// SIMATIC STEP 7 (V5.x) project ZEn01_12_STEP7__Com_SFC2
// program: ProgrammClient(MPI=10) - Example  Communication  SFC XSEND / XRCV
client program
// program: ProgrammServer(MPI=15) - Example communication SFC XSEND / XRCV
server program

SYMBOL_TABLE
"Data_X_SEND-1"	DB 1	DB 1
"Data_X_SEND-2"	DB 2	DB 2
"Data_X_SEND-3"	DB 3	DB 3
"Modify Values"	FC 1	FC 1
"Communication(send)"	FC 10	FC 10
"CYCL_EXC"	OB 1	OB 1	// Cycle Execution
"CYC_INT5"	OB 35	OB 35	// Cyclic Interrupt 5
"COMPLETE RESTART"	OB 100	OB 100	// Complete Restart
"X_SEND"	SFC 65	SFC 65
"X_RCV"	SFC 66	SFC 66
"X_GET"	SFC 67	SFC 67
"X_PUT"	SFC 68	SFC 68
"X_ABORT"	SFC 69	SFC 69
"I_GET"	SFC 72	SFC 72
"I_PUT"	SFC 73	SFC 73
"I_ABORT"	SFC 74	SFC 74
END_SYMBOL_TABLE

FUNCTION "Modify Values" : VOID	// FC 1
TITLE = Function for Generating a Modifiable Date
AUTHOR : SIEMENS
VERSION : 1.0
BEGIN
NETWORK
TITLE = Incrementing and Saving a Value
      L     MD 60;
      L     1;
      +D;
      T     MD 60;
//Save the variables to be sent in a double word
      T     DB1.DBD 0;	//First double word of variable "X_SEND-1".Array10Byte 
      T     "Data_X_SEND-2".DoubleWord;	//Variable "X_SEND-2".DoubleWord
      T     DB3.DBD 0;	//First double word of variable "X_SEND-3".Array3Words
END_FUNCTION

FUNCTION "Communication(send)" : VOID	// FC 10
VERSION : 1.0
BEGIN
NETWORK
TITLE = X_SEND Block Call 
//Query which X_SEND SFC is currently active
      L     MW 50;	//X_SEND SFC variable: "X_SEND-1".Array10Byte (DB1.DBb 0 to 9) 
      L     1;
      ==I;
      JC    m001;	//Jump to SFC X_SEND variable: "X_SEND-1".Array10Byte  
      L     MW 50;	//X_SEND SFC variable: "X_SEND-2".DoubleWord (DB2.DBD 0) 
      L     2;
      ==I;
      JC    m002;	//Jump to X_SEND SFC variable: "X_SEND-2".DoubleWord  
      L     MW 50;	//X_SEND SFC variable: "X_SEND-3".Array3Words (DB1.DBW 0 to 3) 
      L     3;
      ==I;
      JC    m003;	//Jump to X_SEND SFC variable: "X_SEND-3".Array3Words  
      BEU;
m001: CALL  "X_SEND" (
           REQ                      := M 100.2,
           CONT                     := M 100.3,
           DEST_ID                  := MW 110,
           REQ_ID                   := MD 120,
           SD                       := "Data_X_SEND-1".Array10Bytes,
           RET_VAL                  := MW 132,
           BUSY                     := M 100.4);	//Call X_SEND block / Transfer data (Yes/No)? / Maintain connection (Yes/No)? / Address of receiver / Job number / Send data 10 bytes (DB1) / Return value / SFC active?
//Edge evaluation: Is communication with the falling edge of the BUSY bit
//finished?
      A     M 100.4;
      FN    M 100.5;
      JC    m004;	//Jump to increment the communication memory word
      BEU;
m002: CALL  "X_SEND" (
           REQ                      := M 101.2,
           CONT                     := M 101.3,
           DEST_ID                  := MW 112,
           REQ_ID                   := MD 124,
           SD                       := "Data_X_SEND-2".DoubleWord,
           RET_VAL                  := MW 134,
           BUSY                     := M 101.4);	//Call X_SEND block / Transfer data (Yes/No)? / Maintain connection (Yes/No)? / Address of receiver / Job number / Send data 1 double word (DB2) / Return value / SFC active?
//Edge evaluation: Is communication with the falling edge of the BUSY bit
//finished?
      A     M 101.4;
      FN    M 101.5;
      JC    m005;	//Jump to increment the communication memory word
      BEU;
m003: CALL  "X_SEND" (
           REQ                      := M 102.2,
           CONT                     := M 102.3,
           DEST_ID                  := MW 114,
           REQ_ID                   := MD 128,
           SD                       := "Data_X_SEND-3".Array3Words,
           RET_VAL                  := MW 136,
           BUSY                     := M 102.4);	//Call X_SEND block / Transfer data (Yes/No)? / Maintain connection (Yes/No)? / Address of receiver / Job number / Send data 3 words (DB3) / Return value / SFC active?
//Edge evaluation: Is communication with the falling edge of the BUSY bit
//finished?
      A     M 102.4;
      FN    M 102.5;
      JC    m006;	//Jump to increment the communication memory word
      BEU;
//In the following section, the communication counter is incremented following  
//communication.
m004: L     2;	//Increment after sending "X_SEND-1".Array10Byte
      T     MW 50;
      CALL  "Modify Values";	//The values in the variables are incremented
      BEU;
m005: L     3;	//Increment after sending "X_SEND-2".DoubleWord
      T     MW 50;
      CALL  "Modify Values";	//The values in the variables are incremented
      BEU;
m006: L     1;	//Increment after sending "X_SEND-3".Array3Words
      T     MW 50;
      CALL  "Modify Values";	//The values in the variables are incremented
      BEU;
END_FUNCTION

DATA_BLOCK "Data_X_SEND-1"	// DB 1
AUTHOR : SIEMENS
VERSION : 1.0
  STRUCT
   Array10Bytes : ARRAY  [1 .. 10 ] OF //Array of 10 bytes
   BYTE  := 5 (B#16#10) , 5 (B#16#10) ;
  END_STRUCT ;	
BEGIN
   Array10Bytes[1] := B#16#10;
   Array10Bytes[2] := B#16#10;
   Array10Bytes[3] := B#16#10;
   Array10Bytes[4] := B#16#10;
   Array10Bytes[5] := B#16#10;
   Array10Bytes[6] := B#16#10;
   Array10Bytes[7] := B#16#10;
   Array10Bytes[8] := B#16#10;
   Array10Bytes[9] := B#16#10;
   Array10Bytes[10] := B#16#10;
END_DATA_BLOCK

DATA_BLOCK "Data_X_SEND-2"	// DB 2
AUTHOR : SIEMENS
VERSION : 1.0
  STRUCT
   DoubleWord : DWORD  := DW#16#2D;	//Double word
  END_STRUCT ;	
BEGIN
   DoubleWord := DW#16#2D;
END_DATA_BLOCK

DATA_BLOCK "Data_X_SEND-3"	// DB 3
AUTHOR : SIEMENS
VERSION : 1.0
  STRUCT
   Array3Words : ARRAY  [1 .. 3 ] OF //Array of 3 words
   WORD  := 3 (W#16#3) ;
  END_STRUCT ;	
BEGIN
   Array3Words[1] := W#16#3;
   Array3Words[2] := W#16#3;
   Array3Words[3] := W#16#3;
END_DATA_BLOCK

ORGANIZATION_BLOCK "CYCL_EXC"	// OB 1
TITLE = Cyclically Processing Program
AUTHOR : SIEMENS
VERSION : 1.0
VAR_TEMP
  OB1_EV_CLASS : BYTE ;	//Bits 0 to 3 = 1 (incoming event), bits 4 to 7 = 1 (event class 1)
  OB1_SCAN_1 : BYTE ;	//1 (Cold restart scan 1 of OB1), 3 (Scan 2-n of OB1)
  OB1_PRIORITY : BYTE ;	//1 (Priority of 1 is lowest)
  OB1_OB_NUMBR : BYTE ;	//1 (Organization block 1, OB1)
  OB1_RESERVED_1 : BYTE ;	//Reserved for system
  OB1_RESERVED_2 : BYTE ;	//Reserved for system
  OB1_PREV_CYCLE : INT ;	//Cycle time of previous OB1 scan (milliseconds)
  OB1_MIN_CYCLE : INT ;	//Minimum cycle time of OB1 (milliseconds)
  OB1_MAX_CYCLE : INT ;	//Maximum cycle time of OB1 (milliseconds)
  OB1_DATE_TIME : DATE_AND_TIME ;	//Date and time OB1 started
END_VAR
BEGIN
NETWORK
TITLE = Description of the Communication Function 
NETWORK
TITLE = Default Settings for the SFC Parameters
//
//By setting the following 3 memory bits, you can ensure that the connection 
//between 
//the communication partners is retained following each SFC call.
      SET;
      =     M 100.3;	//Connection should be maintained after SFC call 
      =     M 101.3;	//Connection should be maintained after SFC call
      =     M 102.3;	//Connection should be maintained after SFC call 
// Default address for SFCs
      L     15;	//Load MPI subnet address or 
//                                        the address of the logical node number
      T     MW 110;	//SFC call, send an array of 10 bytes (DB1)
      T     MW 112;	//SFC call, send a double word (DB2)
      T     MW 114;	//SFC call, send an array of 3 words (DB3)
//Assignment of the job number
      L     1;	//Load first job number
      T     MD 120;	//Assign to SFC call (array of 10 bytes)
      L     2;	//Load second job number
      T     MD 124;	//Assign to SFC call (double word)
      L     3;	//Load third job number
      T     MD 128;	//Assign to SFC call (array 3 words)
END_ORGANIZATION_BLOCK

ORGANIZATION_BLOCK "CYC_INT5"	// OB 35
TITLE = Call Every 100 ms
AUTHOR : SIEMENS
VERSION : 1.0
VAR_TEMP
  OB35_EV_CLASS : BYTE ;	//Bits 0 to 3 = 1 (incoming event), bits 4 to 7 = 1 (event class 1)
  OB35_STRT_INF : BYTE ;	//16#36 (OB35 has started)
  OB35_PRIORITY : BYTE ;	//11 (Priority of 1 is lowest)
  OB35_OB_NUMBR : BYTE ;	//35 (Organization block 35, OB35)
  OB35_RESERVED_1 : BYTE ;	//Reserved for system
  OB35_RESERVED_2 : BYTE ;	//Reserved for system
  OB35_PHASE_OFFSET : WORD ;	//Phase offset (ms)
  OB35_RESERVED_3 : INT ;	//Reserved for system
  OB35_EXC_FREQ : INT ;	//Frequency of execution (ms)
  OB35_DATE_TIME : DATE_AND_TIME ;	//Date and time OB35 started
END_VAR
BEGIN
NETWORK
TITLE = Communicating with Server S7 Station B
//********************************************************************************
//******************
//General Description of the Communication Function of this Client S7 Station A
//********************************************************************************
//******************
//
//Three variables are exchanged between this client S7-300 station A and the 
//server S7-300 station B. 
//The variable "X_SEND-1".Feld10byte (DB1.DBB 0 to 9) is sent to server MPI 15 
//with the SFC X_SEND.
//An SFC call is required for this.
//The same procedure is required for the variable "X_SEND-2".Doppelwort (DB2.DBD 
//0).
//The variable "X_SEND-1".Feld3Worte (DB3.DBW 0 to 2) is the third variable to be 
//written by the  
//client to a variable of the same name on the server with the SFC X_SEND.
//The variables can be found in DBs 1 to 3 on both the client and the server 
//side. 
//The connection between the communicating CPUs is established the first time an 
//SFC is called 
//and then maintained (only one connection resource is required).
//The SFCs are called by OB35 using a timer in order to make them independent of 
//the 
//scan cycle time of OB1 in the client and the server CPU.
//The timers for the OB calls are preset when the CPU is configured.
//In this CPU, OB35 is called every 100 ms(default), and this means that the 
//various SFCs are also 
//called every 100 ms (max.). 
//Once data exchange is complete, the data are changed in the variables in order 
//to show that  
//data have been received. If there is an error in the communication, and no data 
//are
//sent, the data in the receiver will not change. 
//If the receive data are continually changing, this means that data exchange is 
//taking place. 
//
//
//Note:
//The memory words in which the RET_VALS of the SFCs are entered should be 
//evaluated while the  
//program is running. If an SFC registers an error value, it can still be 
//correctly executed, 
//although no data will have been sent. 
//As soon as the RET_VAL of an SFC becomes negative, this signals that an error 
//has
//occurred during data transmission. 
//
//
//Memory words in which the RET_VALs are entered:
//MW130, MW132, MW134
//
//The above note was not taken into account in this programming example, since 
//error messages 
//which may occur cannot be converted to corresponding messages (alarms which 
//appear on the device) 
//until a real control program is run.
//
      CALL  "Communication(send)";	//Call communication function
END_ORGANIZATION_BLOCK

ORGANIZATION_BLOCK "COMPLETE RESTART"	// OB 100
AUTHOR : SIEMENS
VERSION : 1.0
VAR_TEMP
  OB100_EV_CLASS : BYTE ;	//16#13, Event class 1, entering event state, event logged in diagnostic buffer
  OB100_STRTUP : BYTE ;	//16#81/82/83/84 Method of startup
  OB100_PRIORITY : BYTE ;	//27 (Priority of 1 is lowest)
  OB100_OB_NUMBR : BYTE ;	//100 (Organization block 100, OB100)
  OB100_RESERVED_1 : BYTE ;	//Reserved for system
  OB100_RESERVED_2 : BYTE ;	//Reserved for system
  OB100_STOP : WORD ;	//Event that caused CPU to stop (16#4xxx)
  OB100_STRT_INFO : DWORD ;	//Information on how system started
  OB100_DATE_TIME : DATE_AND_TIME ;	//Date and time OB100 started
END_VAR
BEGIN
NETWORK
TITLE = Initial Value Assignment
      L     1;	//Preset communication memory word
      T     MW 50;
      SET;	//Set starting memory bit of SFC X_SEND   
      =     M 100.2;	//SFC X_SEND variable: "X_SEND-1".Array10Byte
      =     M 101.2;	//SFC X_SEND variable: "X_SEND-2".DoubleWord
      =     M 102.2;	//SFC X_SEND variable: "X_SEND-3".Array3Words
END_ORGANIZATION_BLOCK

SYMBOL_TABLE
"Data_X_RCV-1"	DB 1	DB 1
"Data_X_RCV-2"	DB 2	DB 2
"Data_X_RCV-3"	DB 3	DB 3
"Modify Values"	FC 1	FC 1
"Communication(receive)"	FC 20	FC 20
"CYCL_EXC"	OB 1	OB 1	// Cycle Execution
"CYC_INT5"	OB 35	OB 35	// Cyclic Interrupt 5
"COMPLETE RESTART"	OB 100	OB 100	// Complete Restart
"X_SEND"	SFC 65	SFC 65
"X_RCV"	SFC 66	SFC 66
"X_GET"	SFC 67	SFC 67
"X_PUT"	SFC 68	SFC 68
"X_ABORT"	SFC 69	SFC 69
"I_GET"	SFC 72	SFC 72
"I_PUT"	SFC 73	SFC 73
"I_ABORT"	SFC 74	SFC 74
END_SYMBOL_TABLE

FUNCTION "Communication(receive)" : VOID	// FC 20
TITLE = Receiving Data from Client S7 Station A
AUTHOR : SIEMENS
VERSION : 1.0
VAR_TEMP
  NIL_PTR : ANY ;	//NIL pointer, required in order to discard data
END_VAR
BEGIN
NETWORK
TITLE = Call X_RCV Block
//OB35 is called by the operating system every 100 ms (any value higher or lower  
//than this can be selected). FC20 is called in OB35. 
//The job number of the incoming data assigned by the sender is determined in FC20
//when X_RCV (SFC66) is first called. 
//This sender job number is then used to assign the data received to the 
//corresponding 
//data area and to copy them to this area when X_RCV is called again.
//
//
//If the receive data are not evaluated for any reason, they must be 
//removed from the receive buffer and written to a NIL pointer.
//The following section of this network contains the branch instruction which
//determines whether the data are received or discarded.
//
      JU    add;	//Jump to accept the receive data
//    SPA   disc                        //Jump to discard the receive data
      BEU;
add:  CLR;
      =     M 100.2;	//Reset the data accept memory bit
      CALL  "X_RCV" (
           EN_DT                    := M 100.2,
           RET_VAL                  := MW 130,
           REQ_ID                   := MD 120,
           NDA                      := M 100.5,
           RD                       := "Data_X_RCV-1".Array10Bytes);	//Call receive SFC for evaluation / Accept data (Yes/No)? / Return value / Job number of sender / Receive new data? / Receive data area
      A     M 100.5;	//Have new data been received?
      JC    Case;	//If data have been received, call SFC again and
//                                        add data to user area
      BEU;	//Block end absolute
Case: L     MD 120;	//Load job number of sender
      L     1;	//Compare with job number 1
      ==I;
      JC    add1;	//Jump to accept data
      L     MD 120;	//Load job number of sender
      L     2;	//Compare with job number 2
      ==I;
      JC    add2;	//Jump to accept data
      L     MD 120;	//Load job number of sender
      L     3;	//Compare with job number 3
      ==I;
      JC    add3;	//Jump to accept data
      JU    end;	//Jump to network end
add1: SET;	//Set RLO = 1 to add data to target area
      =     M 100.2;
      CALL  "X_RCV" (
           EN_DT                    := M 100.2,
           RET_VAL                  := MW 132,
           REQ_ID                   := MD 124,
           NDA                      := M 101.5,
           RD                       := "Data_X_RCV-1".Array10Bytes);	//Call receive SFC to accept data / Accept data? / Return value / Job number / Receive new data? / Selected receive data area DB1 (variable size: 10 bytes)
      JU    end;	//Jump to network end
add2: SET;	//Set RLO = 1 to add data to target area
      =     M 100.2;
      CALL  "X_RCV" (
           EN_DT                    := M 100.2,
           RET_VAL                  := MW 132,
           REQ_ID                   := MD 124,
           NDA                      := M 101.5,
           RD                       := "Data_X_RCV-2".DoubleWord);	//Call receive SFC to accept data / Accept data? / Return value / Job number / Receive new data? / Selected receive data area DB2 (variable size: 1 double word)
      JU    end;	//Jump to network end
add3: SET;	//Set RLO = 1 to add data to target area
      =     M 100.2;
      CALL  "X_RCV" (
           EN_DT                    := M 100.2,
           RET_VAL                  := MW 132,
           REQ_ID                   := MD 124,
           NDA                      := M 101.5,
           RD                       := "Data_X_RCV-3".Array3Words);	//Call receive SFC to accept data / Accept data? / Return value / Job number / Receive new data? / Selected receive data area DB3 (variable size: 3 words)
end:  NOP   0;	//Network end
      BEU;
NETWORK
TITLE = Discarding the Receive Data
//disc: NOP   1                         //This line must be added if the receive 
//data are to be
//                                        discarded with the NIL pointer.
// (network holds code this reader does not know; not shown)
END_FUNCTION

DATA_BLOCK "Data_X_RCV-1"	// DB 1
AUTHOR : SIEMENS
VERSION : 1.0
  STRUCT
   Array10Bytes : ARRAY  [1 .. 10 ] OF //Array of 10 bytes
   BYTE  := 5 (B#16#10) , 5 (B#16#10) ;
  END_STRUCT ;	
BEGIN
   Array10Bytes[1] := B#16#10;
   Array10Bytes[2] := B#16#10;
   Array10Bytes[3] := B#16#10;
   Array10Bytes[4] := B#16#10;
   Array10Bytes[5] := B#16#10;
   Array10Bytes[6] := B#16#10;
   Array10Bytes[7] := B#16#10;
   Array10Bytes[8] := B#16#10;
   Array10Bytes[9] := B#16#10;
   Array10Bytes[10] := B#16#10;
END_DATA_BLOCK

DATA_BLOCK "Data_X_RCV-2"	// DB 2
AUTHOR : SIEMENS
VERSION : 1.0
  STRUCT
   DoubleWord : DWORD  := DW#16#2D;	//Double word
  END_STRUCT ;	
BEGIN
   DoubleWord := DW#16#2D;
END_DATA_BLOCK

DATA_BLOCK "Data_X_RCV-3"	// DB 3
AUTHOR : SIEMENS
VERSION : 1.0
  STRUCT
   Array3Words : ARRAY  [1 .. 3 ] OF //Array of 3 words
   WORD  := 3 (W#16#3) ;
  END_STRUCT ;	
BEGIN
   Array3Words[1] := W#16#3;
   Array3Words[2] := W#16#3;
   Array3Words[3] := W#16#3;
END_DATA_BLOCK

ORGANIZATION_BLOCK "CYCL_EXC"	// OB 1
TITLE = "Main Program Sweep (Cycle)"
VERSION : 0.0
VAR_TEMP
  OB1_EV_CLASS : BYTE ;	//Bits 0-3 = 1 (Coming event), Bits 4-7 = 1 (Event class 1)
  OB1_SCAN_1 : BYTE ;	//1 (Cold restart scan 1 of OB 1), 3 (Scan 2-n of OB 1)
  OB1_PRIORITY : BYTE ;	//1 (Priority of 1 is lowest)
  OB1_OB_NUMBR : BYTE ;	//1 (Organization block 1, OB1)
  OB1_RESERVED_1 : BYTE ;	//Reserved for system
  OB1_RESERVED_2 : BYTE ;	//Reserved for system
  OB1_PREV_CYCLE : INT ;	//Cycle time of previous OB1 scan (milliseconds)
  OB1_MIN_CYCLE : INT ;	//Minimum cycle time of OB1 (milliseconds)
  OB1_MAX_CYCLE : INT ;	//Maximum cycle time of OB1 (milliseconds)
  OB1_DATE_TIME : DATE_AND_TIME ;	//Date and time OB1 started
END_VAR
BEGIN
NETWORK
TITLE =
END_ORGANIZATION_BLOCK

ORGANIZATION_BLOCK "CYC_INT5"	// OB 35
TITLE = Call Every 100 ms
AUTHOR : SIEMENS
VERSION : 1.0
VAR_TEMP
  OB35_EV_CLASS : BYTE ;	//Bits 0 to 3 = 1 (incoming event), bits 4 to 7 = 1 (event class 1)
  OB35_STRT_INF : BYTE ;	//16#36 (OB35 has started)
  OB35_PRIORITY : BYTE ;	//11 (Priority of 1 is lowest)
  OB35_OB_NUMBR : BYTE ;	//35 (Organization block 35, OB35)
  OB35_RESERVED_1 : BYTE ;	//Reserved for system
  OB35_RESERVED_2 : BYTE ;	//Reserved for system
  OB35_PHASE_OFFSET : WORD ;	//Phase offset (ms)
  OB35_RESERVED_3 : INT ;	//Reserved for system
  OB35_EXC_FREQ : INT ;	//Frequency of execution (ms)
  OB35_DATE_TIME : DATE_AND_TIME ;	//Date and time OB35 started
END_VAR
BEGIN
NETWORK
TITLE = Timer-Controlled Call of Data Receive Function
//Description of the Communication Function of Server
//********************************************************************************
//****
//General Description of the Communication Function of this CPU
//********************************************************************************
//****
//In OB35, which is called every 100 ms by the CPU, several X_RCV SFCs are called 
//using different receive address areas. 
//The data come from the client CPU and are stored here in the variables 
//["X_SEND-1".Feld10byte (db1.dbb 0 to 9)], ["X_SEND-2".Doppelwort (db2.dbb 0)],  
//and ["X_SEND-3".Feld3Worte (db3.dbw 0 to 2)].
//The incoming variables are received by an SFC X_RCV and, depending on their job 
//number, stored in the correct data area of the server.
//Using the Monitor Variable function in VAT1 of this server CPU, you can 
//monitor the parameters of SFC X_RCV, and the data areas to which the receive 
//data
//are copied are also displayed.
//If these variables are received by the server, you can determine whether a  
//relatively long data exchange is taking place by viewing how the variable 
//contents   
//change, or whether there is any exchange of data at all (if there is no visible 
//change in the variable contents). Using VAT1 (Monitor Variable), you can 
//monitor all 
//the important parameters and the contents of the variables.
      CALL  "Communication(receive)";	//Accept receive data
END_ORGANIZATION_BLOCK

ORGANIZATION_BLOCK "COMPLETE RESTART"	// OB 100
TITLE = "Complete Restart"
VERSION : 0.0
VAR_TEMP
  OB100_EV_CLASS : BYTE ;	//16#13, Event class 1, Entering event state, Event logged in diagnostic buffer
  OB100_STRTUP : BYTE ;	//16#81/82/83/84 Method of startup
  OB100_PRIORITY : BYTE ;	//27 (Priority of 1 is lowest)
  OB100_OB_NUMBR : BYTE ;	//100 (Organization block 100, OB100)
  OB100_RESERVED_1 : BYTE ;	//Reserved for system
  OB100_RESERVED_2 : BYTE ;	//Reserved for system
  OB100_STOP : WORD ;	//Event that caused CPU to stop (16#4xxx)
  OB100_STRT_INFO : DWORD ;	//Information on how system started
  OB100_DATE_TIME : DATE_AND_TIME ;	//Date and time OB100 started
END_VAR
BEGIN
NETWORK
TITLE =
END_ORGANIZATION_BLOCK
